{attribute 'GeneratedUsingTerminal: EL3773-0000-0019'}
{attribute addProperty BoxType "EL3773-0000-0019"}
{attribute addProperty Id "I2_SamplesAT %I*I2_Samples_2549228720"}
{attribute addProperty CRC "2864058222"}
{attribute addProperty Size "20"}
TYPE L2_Current_Samples_AAB60F6E :
STRUCT
	{attribute addProperty Name "I2_Samples"}
	I2_Samples AT %I* : I2_Samples_25492287;
END_STRUCT
END_TYPE

(* stored: Version 1.2.0.0, ProductVersion 3.1.4024.9
   DUT L2_Current_Samples_AAB60F6E: Id {90b575c6-c5fa-4944-9529-c3c8733fb2c8} *)
